// TwinCAT 3 PLC project PLCPrg
// ProgramVersion: 3.1.4024.0
// libraries:
//   Tc2_MC2, * (Beckhoff Automation GmbH)
//   Tc2_Standard, * (Beckhoff Automation GmbH)
//   Tc2_System, * (Beckhoff Automation GmbH)
//   Tc3_Module, * (Beckhoff Automation GmbH)
// project tree:
//   / PlcTask.TcTTO
//   POUs/Axis/ AxisConfigurationO.TcDUT, MotionAxisO.TcPOU
//   POUs/ MAIN.TcPOU, OOPSDevelopmentTest.TcPOU, OOPSOld.TcPOU
// real-time tasks:
//   TASK PlcTask: cycle T#10ms, priority 20, ADS port 350
// motion (NC):
//   TASK Motion SAF: cycle T#2ms, priority 4, ADS port 501
//   TASK Motion SVB: cycle T#10ms, priority 8, ADS port 511
//   AXIS Axis 1 (id 1)
//     OtherSettings: AllowMotionCmdToSlave=true
//     encoder EncType=1
//     drive DrvType=5
//       Analog: TorqueSetpointScale=10, ScaleFactorActTorque=0.1
//       TimeComp: TaskDelayCycles=1
//     controller CtrType=1
//       CtrPara: PriorControlFactor=1
//         Observer: BandWidth=20
// I/O:
//   DEVICE Device 1 (EtherCAT), AmsNetId 192.168.0.50.2.1
//     Term 1 (EK1100) [EK1100 EtherCAT Coupler (2A E-Bus)]
//       Term 2 (EL2535-0005) [EL2535-0005 2Ch. Pulse Width Current Output (24V, 5 A)]
// variable links:
//   PLCPrg/PLCPrg Instance <-> Motion SAF/Axes/Axis 1
//     PlcTask Inputs/MAIN.testAxis.axisRef.NcToPlc <-> Outputs/ToPlc
//     PlcTask Outputs/MAIN.testAxis.axisRef.PlcToNc <-> Inputs/FromPlc

CONFIGURATION PLCPrg
    RESOURCE PLC ON TwinCAT3
        TASK PlcTask(INTERVAL := T#10ms, PRIORITY := 20);
        PROGRAM MAIN WITH PlcTask : MAIN;
    END_RESOURCE
END_CONFIGURATION

// ---- POUs/Axis/AxisConfigurationO.TcDUT
TYPE AxisConfigurationO :
STRUCT
	(* Axis Enable Setting *)
	Override : REAL := 100.0;
	EnablePositive : BOOL:=TRUE;
	EnableNegative : BOOL:=TRUE;
	
	(* Jog Setting *)
	JogMode : E_JogMode:=E_JogMode.MC_JOGMODE_INCHING;
	JogInchingPosition : LREAL:=10.0;
	JogVelocity : LREAL:=100.0;
	JogAccleration : LREAL:=1000.0;
	JogDeaccleration : LREAL:=1000.0;
END_STRUCT
END_TYPE

// ---- POUs/MAIN.TcPOU
PROGRAM MAIN
VAR

END_VAR

//Old
OOPSOld();

//Under Developement
OOPSDevelopmentTest();

END_PROGRAM

// ---- POUs/OOPSOld.TcPOU
PROGRAM OOPSOld
VAR
	testAxis : MotionAxisO;
	AxisEnable: BOOL;
	AxisDisable: BOOL;
	state: BOOL;
	erroID:UDINT;
	pos:LREAL;
	vel:LREAL;
	JogFwd: BOOL;
	JogRev:BOOL;
	modess: E_JogMode;
	testconfig: AxisConfigurationO;
END_VAR

//Test Axis Config
testAxis.configure(stAxisConfig:=testconfig);

//Enable
IF AxisEnable THEN
	testAxis.Enable();
END_IF

IF AxisDisable THEN
	testAxis.Disable();
END_IF

//Jog Method 
testAxis.Jog(JogFrw:=JogFwd,JogRev:=JogRev);


//
state := testAxis.AxisState;
erroID:=testAxis.ErrorID;
pos:=testAxis.ActualPosition;
vel:=testAxis.ActualSpeed;

END_PROGRAM

// ---- POUs/Axis/MotionAxisO.TcPOU
FUNCTION_BLOCK MotionAxisO
VAR
	(* Axis Reference *)
	axisRef : AXIS_REF; 
	
	(* Motion Function Block *)
	fbMcPower 		: MC_Power;				// FB for enable and override
	fbMcReset 		: MC_Reset;				// FB to reset axis
	fbMcStop 		: MC_Stop;				// FB to stop axis
	fbMcHalt		: MC_Halt;				// FB to halt axis
	fbMcMoveAbsolute: MC_MoveAbsolute;		// FB to move axis (Absolute Move)
	fbMcMoveRelative: MC_MoveRelative;		// FB to move axis (Relative Move)
	fbMcJog         : MC_Jog;				// FB to move axis (Relative Move)
	
	(* Axis Config Settings *)
	axisConfig : AxisConfigurationO;
	
	(* Axis Status *)
	axisStatus : BOOL;
	blockError : BOOL;
	nErrorID	   : UDINT;

END_VAR

METHOD AbsoluteMove : BOOL
VAR_INPUT
	TargetPosition : LREAL;
END_VAR

VAR
END_VAR
END_METHOD

PROPERTY ActualPosition : LReal
GET
ActualPosition := axisRef.NcToPlc.ActPos;
END_GET
END_PROPERTY

PROPERTY ActualSpeed : LReal
GET
ActualSpeed := axisRef.NcToPlc.ActVelo;
END_GET
END_PROPERTY

PROPERTY AxisState : BOOL
GET
AxisState:= axisRef.NcToPlc.StateDWord.0 AND axisStatus ;
END_GET
END_PROPERTY

METHOD configure :BOOL;
VAR_INPUT
	stAxisConfig : AxisConfigurationO;
END_VAR
axisConfig := stAxisConfig;

//Not Implemented
configure:=TRUE;
END_METHOD

METHOD Disable : BOOL
VAR
END_VAR
Disable := mcPower(enable:=FALSE);
END_METHOD

METHOD Enable : BOOL
VAR
END_VAR
Enable := mcPower(enable:=TRUE);
END_METHOD

PROPERTY Error : Bool
GET
Error := axisRef.NcToPlc.StateDWord.31 OR blockError;
END_GET
END_PROPERTY

PROPERTY ErrorID : UDINT
GET
ErrorID := nErrorID;
END_GET
END_PROPERTY

METHOD Jog : BOOL;
VAR_INPUT
	JogFrw : BOOL;
	JogRev : BOOL;
END_VAR
Jog := mcJog(jogFrw:=JogFrw,jogRev:=JogRev);
END_METHOD

METHOD INTERNAL mcJog : BOOL
VAR_INPUT
	jogFrw : BOOL;
	jogRev : BOOL;
END_VAR
(* Jog Frw/Rev *)
fbMcJog(
		Axis:=axisRef, 
		JogForward:=jogFrw, 
		JogBackwards:=jogRev, 
		Mode:=axisConfig.JogMode, 
		Position:=axisConfig.JogInchingPosition, 
		Velocity:=axisConfig.JogVelocity, 
		Acceleration:=axisConfig.JogAccleration, 
		Deceleration:=axisConfig.JogDeaccleration);
		
(* Error Handling *)
IF fbMcJog.Error THEN
	blockError:= TRUE;
	nErrorID := fbMcJog.ErrorID;
END_IF

(* Jog State *)
mcJog := fbMcJog.Active;
END_METHOD

METHOD mcMoveAbs : BOOL
VAR_INPUT
	TargetPosition : LREAL;
END_VAR

VAR
	previousTargetPosition : LREAL;
END_VAR
(* Absloute Move *)
IF TargetPosition <> previousTargetPosition THEN
	
END_IF

(* Absloute Move Block *)
fbMcMoveAbsolute(
				Axis:= axisRef, 
				Execute:= , 
				Position:= , 
				Velocity:= , 
				Acceleration:= , 
				Deceleration:= , 
				Jerk:= , 
				BufferMode:= , 
				Options:= , 
				Done=> , 
				Busy=> , 
				Active=> , 
				CommandAborted=> , 
				Error=> , 
				ErrorID=> );
		
(* Error Handling *)
IF fbMcMoveAbsolute.Error THEN
	blockError:= TRUE;
	nErrorID := fbMcMoveAbsolute.ErrorID;
END_IF

(* Absolute Move Complete *)
mcMoveAbs := fbMcMoveAbsolute.Done AND NOT fbMcMoveAbsolute.Busy ;
END_METHOD

METHOD INTERNAL mcPower : BOOL
VAR_INPUT
	enable : BOOL;
END_VAR
(* Axis Enable/Disable *)
fbMCPower(Enable 			:= enable, 
		  Enable_Positive	:= axisConfig.EnablePositive, 
		  Enable_Negative	:= axisConfig.EnableNegative, 
		  Override		    := axisConfig.Override,
	      Axis			    := axisRef);

(* Error Handling *)
IF fbMcPower.Error THEN
	blockError:= TRUE;
	nErrorID := fbMcPower.ErrorID;
END_IF

(* Axis State *)
mcPower := axisStatus := fbMCPower.Status;
END_METHOD

END_FUNCTION_BLOCK

// ---- POUs/OOPSDevelopmentTest.TcPOU
PROGRAM OOPSDevelopmentTest
VAR
END_VAR

END_PROGRAM
